FUNCTION_BLOCK FB_JsonLogger EXTENDS FB_AbstractLogger
VAR
	sJson:					STRING(1000);
	JsonDocument: 			SJsonValue;
	fbJsonParser:			FB_JsonDomParser;
END_VAR

// https://github.com/PeterZerlauth/Tc3_Component
IF TwinCAT_SystemInfoVarList._TaskInfo[GETCURTASKINDEXEX()].FirstCycle THEN
	jsonDocument:= fbJsonParser.NewDocument();
	fbJsonParser.CopyString(jsonDocument, sJson, SIZEOF(sJson));
END_IF

METHOD PUBLIC M_Insert : SJsonValue
VAR_INPUT
	sJson:			STRING(255);
END_VAR
// Find event in buffer
M_Insert := fbJsonParser.AddArrayMember(JsonDocument, sJson, 0);

fbJsonParser.CopyString(jsonDocument, sJson, SIZEOF(sJson));
END_METHOD

METHOD PUBLIC M_Find : SJsonValue
VAR_INPUT
	sJson:			STRING(255);
END_VAR
// Find event in buffer
M_Find := fbJsonParser.FindMember(jsonDocument, sJson);
END_METHOD

METHOD PUBLIC M_Reset
VAR_INPUT
END_VAR
END_METHOD

METHOD PUBLIC M_Notify
VAR_INPUT
	stEvent:		ST_Event;
END_VAR
VAR 
	sJson:			STRING:= '{Json:"Value"}';
END_VAR
IF M_Find(sJson) = 0 THEN
	M_Insert(sJson);
END_IF
END_METHOD

METHOD PUBLIC M_Delete : BOOL
VAR_INPUT
	nIndex: 			DINT;
END_VAR
END_METHOD

END_FUNCTION_BLOCK

(* stored: Version 1.1.0.1
   POU FB_JsonLogger: Id {3156b304-db8f-03fb-27b7-7c2ee4999221}, SpecialFunc None
   Method M_Insert: Id {44680086-a137-069c-1fcc-b6f0a7f7e714}
   Method M_Find: Id {4d605ea0-e820-08a5-288f-d51ab8e979bd}
   Method M_Reset: Id {9f4eebcc-54dc-002d-0608-dc133ca553aa}
   Method M_Notify: Id {a42c86be-34f4-0425-1584-9e202f4b9155}
   Method M_Delete: Id {ad9cb8bd-6ad9-0fe9-16a5-daa4bac483ff} *)
